FUNCTION_BLOCK FB_SerCom
VAR 	

END_VAR

END_FUNCTION_BLOCK

(* stored: Version 1.1.0.1
   POU FB_SerCom: Id {3deb06f9-a97a-44b7-9d0f-8f0d97e3406b}, SpecialFunc None *)
